% RSLogix 500 project I2P Hands-On 4 - Tyler_Vogt.RSS, saved by version 10.00.00.00 %
PROJECT "UNTITLED"    % processor: Bul.1763 MicroLogix 1100 Series B %

PROGRAM FILES
  LAD 2   14 rungs

DATA FILES
  O0 OUTPUT  4 elements
  I1 INPUT  6 elements
  S2 STATUS  66 elements
  B3 BINARY  1 elements
  T4 TIMER  1 elements
  C5 COUNTER  1 elements
  R6 CONTROL  1 elements
  N7 INTEGER  1 elements
  F8 FLOAT  1 elements

LADDER 2
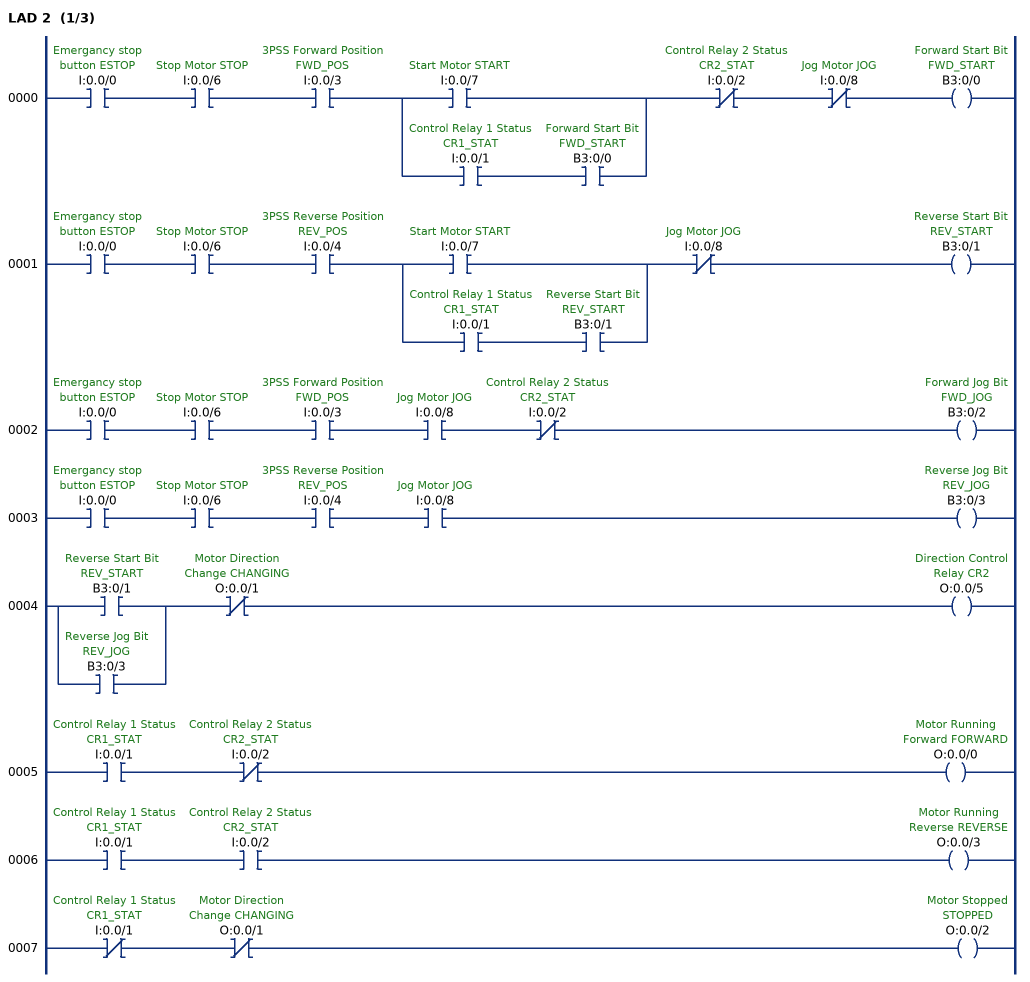
% Rung: 0 %
SOR XIC I:0.0/0 XIC I:0.0/6 XIC I:0.0/3 BST XIC I:0.0/7 NXB XIC I:0.0/1 XIC B3:0/0 BND XIO I:0.0/2 XIO I:0.0/8 OTE B3:0/0 EOR
%   I:0.0/0  ESTOP  "Emergancy stop button" %
%   I:0.0/6  STOP  "Stop Motor" %
%   I:0.0/3  FWD_POS  "3PSS Forward Position" %
%   I:0.0/7  START  "Start Motor" %
%   I:0.0/1  CR1_STAT  "Control Relay 1 Status" %
%   B3:0/0  FWD_START  "Forward Start Bit" %
%   I:0.0/2  CR2_STAT  "Control Relay 2 Status" %
%   I:0.0/8  JOG  "Jog Motor" %
% Rung: 1 %
SOR XIC I:0.0/0 XIC I:0.0/6 XIC I:0.0/4 BST XIC I:0.0/7 NXB XIC I:0.0/1 XIC B3:0/1 BND XIO I:0.0/8 OTE B3:0/1 EOR
%   I:0.0/0  ESTOP  "Emergancy stop button" %
%   I:0.0/6  STOP  "Stop Motor" %
%   I:0.0/4  REV_POS  "3PSS Reverse Position" %
%   I:0.0/7  START  "Start Motor" %
%   I:0.0/1  CR1_STAT  "Control Relay 1 Status" %
%   B3:0/1  REV_START  "Reverse Start Bit" %
%   I:0.0/8  JOG  "Jog Motor" %
% Rung: 2 %
SOR XIC I:0.0/0 XIC I:0.0/6 XIC I:0.0/3 XIC I:0.0/8 XIO I:0.0/2 OTE B3:0/2 EOR
%   I:0.0/0  ESTOP  "Emergancy stop button" %
%   I:0.0/6  STOP  "Stop Motor" %
%   I:0.0/3  FWD_POS  "3PSS Forward Position" %
%   I:0.0/8  JOG  "Jog Motor" %
%   I:0.0/2  CR2_STAT  "Control Relay 2 Status" %
%   B3:0/2  FWD_JOG  "Forward Jog Bit" %
% Rung: 3 %
SOR XIC I:0.0/0 XIC I:0.0/6 XIC I:0.0/4 XIC I:0.0/8 OTE B3:0/3 EOR
%   I:0.0/0  ESTOP  "Emergancy stop button" %
%   I:0.0/6  STOP  "Stop Motor" %
%   I:0.0/4  REV_POS  "3PSS Reverse Position" %
%   I:0.0/8  JOG  "Jog Motor" %
%   B3:0/3  REV_JOG  "Reverse Jog Bit" %
% Rung: 4 %
SOR BST XIC B3:0/1 NXB XIC B3:0/3 BND XIO O:0.0/1 OTE O:0.0/5 EOR
%   B3:0/1  REV_START  "Reverse Start Bit" %
%   B3:0/3  REV_JOG  "Reverse Jog Bit" %
%   O:0.0/1  CHANGING  "Motor Direction Change" %
%   O:0.0/5  CR2  "Direction Control Relay" %
% Rung: 5 %
SOR XIC I:0.0/1 XIO I:0.0/2 OTE O:0.0/0 EOR
%   I:0.0/1  CR1_STAT  "Control Relay 1 Status" %
%   I:0.0/2  CR2_STAT  "Control Relay 2 Status" %
%   O:0.0/0  FORWARD  "Motor Running Forward" %
% Rung: 6 %
SOR XIC I:0.0/1 XIC I:0.0/2 OTE O:0.0/3 EOR
%   I:0.0/1  CR1_STAT  "Control Relay 1 Status" %
%   I:0.0/2  CR2_STAT  "Control Relay 2 Status" %
%   O:0.0/3  REVERSE  "Motor Running Reverse" %
% Rung: 7 %
SOR XIO I:0.0/1 XIO O:0.0/1 OTE O:0.0/2 EOR
%   I:0.0/1  CR1_STAT  "Control Relay 1 Status" %
%   O:0.0/1  CHANGING  "Motor Direction Change" %
%   O:0.0/2  STOPPED  "Motor Stopped" %

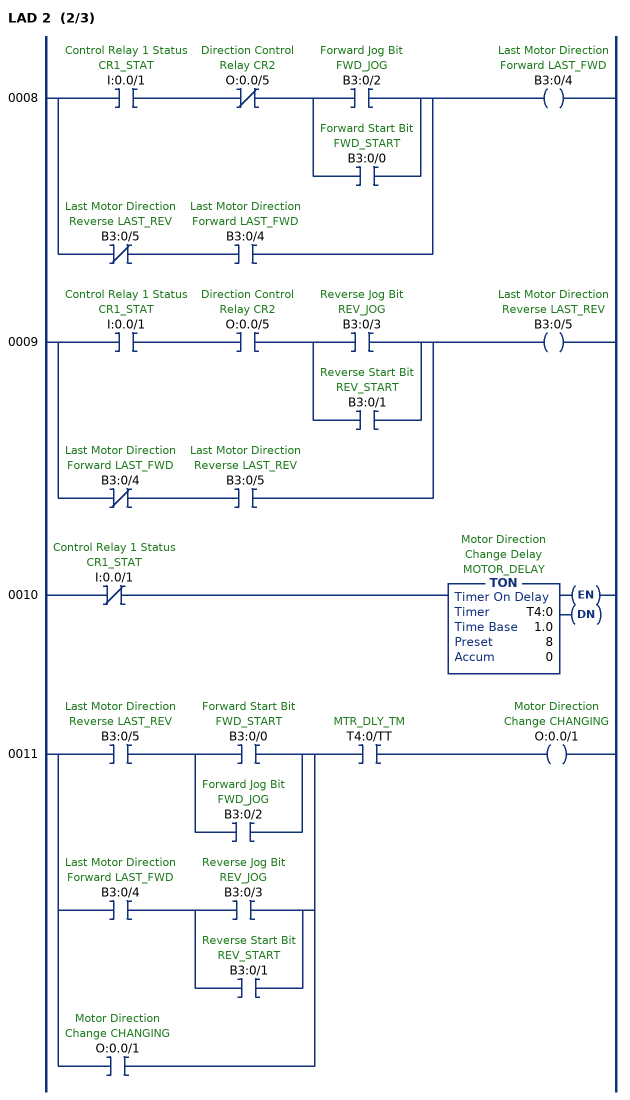
% Rung: 8 %
SOR BST XIC I:0.0/1 XIO O:0.0/5 BST XIC B3:0/2 NXB XIC B3:0/0 BND NXB XIO B3:0/5 XIC B3:0/4 BND OTE B3:0/4 EOR
%   I:0.0/1  CR1_STAT  "Control Relay 1 Status" %
%   O:0.0/5  CR2  "Direction Control Relay" %
%   B3:0/2  FWD_JOG  "Forward Jog Bit" %
%   B3:0/0  FWD_START  "Forward Start Bit" %
%   B3:0/5  LAST_REV  "Last Motor Direction Reverse" %
%   B3:0/4  LAST_FWD  "Last Motor Direction Forward" %
% Rung: 9 %
SOR BST XIC I:0.0/1 XIC O:0.0/5 BST XIC B3:0/3 NXB XIC B3:0/1 BND NXB XIO B3:0/4 XIC B3:0/5 BND OTE B3:0/5 EOR
%   I:0.0/1  CR1_STAT  "Control Relay 1 Status" %
%   O:0.0/5  CR2  "Direction Control Relay" %
%   B3:0/3  REV_JOG  "Reverse Jog Bit" %
%   B3:0/1  REV_START  "Reverse Start Bit" %
%   B3:0/4  LAST_FWD  "Last Motor Direction Forward" %
%   B3:0/5  LAST_REV  "Last Motor Direction Reverse" %
% Rung: 10 %
SOR XIO I:0.0/1 TON T4:0 1.0 8 0 EOR
%   I:0.0/1  CR1_STAT  "Control Relay 1 Status" %
%   T4:0  MOTOR_DELAY  "Motor Direction Change Delay" %
% Rung: 11 %
SOR BST XIC B3:0/5 BST XIC B3:0/0 NXB XIC B3:0/2 BND NXB BST XIC B3:0/4 BST XIC B3:0/3 NXB XIC B3:0/1 BND NXB XIC O:0.0/1 BND BND XIC T4:0/TT OTE O:0.0/1 EOR
%   B3:0/5  LAST_REV  "Last Motor Direction Reverse" %
%   B3:0/0  FWD_START  "Forward Start Bit" %
%   B3:0/2  FWD_JOG  "Forward Jog Bit" %
%   B3:0/4  LAST_FWD  "Last Motor Direction Forward" %
%   B3:0/3  REV_JOG  "Reverse Jog Bit" %
%   B3:0/1  REV_START  "Reverse Start Bit" %
%   O:0.0/1  CHANGING  "Motor Direction Change" %
%   T4:0/TT  MTR_DLY_TM %

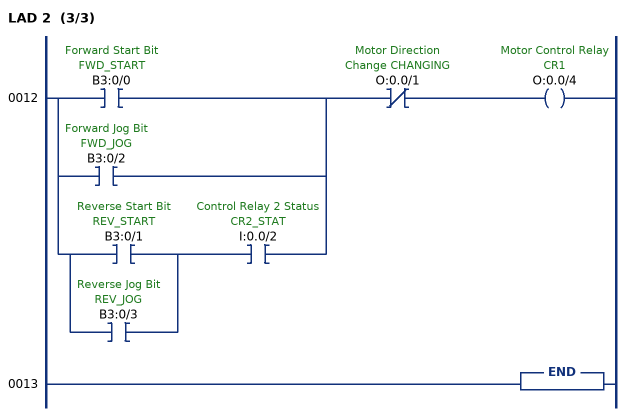
% Rung: 12 %
SOR BST BST XIC B3:0/0 NXB XIC B3:0/2 BND NXB BST XIC B3:0/1 NXB XIC B3:0/3 BND XIC I:0.0/2 BND XIO O:0.0/1 OTE O:0.0/4 EOR
%   B3:0/0  FWD_START  "Forward Start Bit" %
%   B3:0/2  FWD_JOG  "Forward Jog Bit" %
%   B3:0/1  REV_START  "Reverse Start Bit" %
%   B3:0/3  REV_JOG  "Reverse Jog Bit" %
%   I:0.0/2  CR2_STAT  "Control Relay 2 Status" %
%   O:0.0/1  CHANGING  "Motor Direction Change" %
%   O:0.0/4  CR1  "Motor Control Relay" %
% Rung: 13 %
SOR END EOR

DATA TABLE (non-zero values as saved)
DATA T4
% .PRE .ACC %
% T4:0 % 8 0
